// TIA Portal V18 export
// export: Created 2026-06-23T08:49:31.4351033Z, ExportSetting WithDefaults, DisplayName Totally Integrated Automation Portal, DisplayVersion V18, DisplayName TIA Portal Openness, DisplayVersion V18, DisplayName TIA Portal Version Control Interface, DisplayVersion V18, DisplayName STEP 7 Professional, DisplayVersion V18, DisplayName STEP 7 Safety, DisplayVersion V18, DisplayName WinCC Professional, DisplayVersion V18
FUNCTION "FC_HMI_Mirror_PLC2" : Void   // FC41, LAD
{ S7_Optimized_Access := 'TRUE' }
VERSION : 0.1
// stored: AutoNumber true, IsIECCheckEnabled false, SetENOAutomatically false, UDAEnableTagReadback false
BEGIN

REGION Network 1: Mirror V3240_Nuoc_Bon3
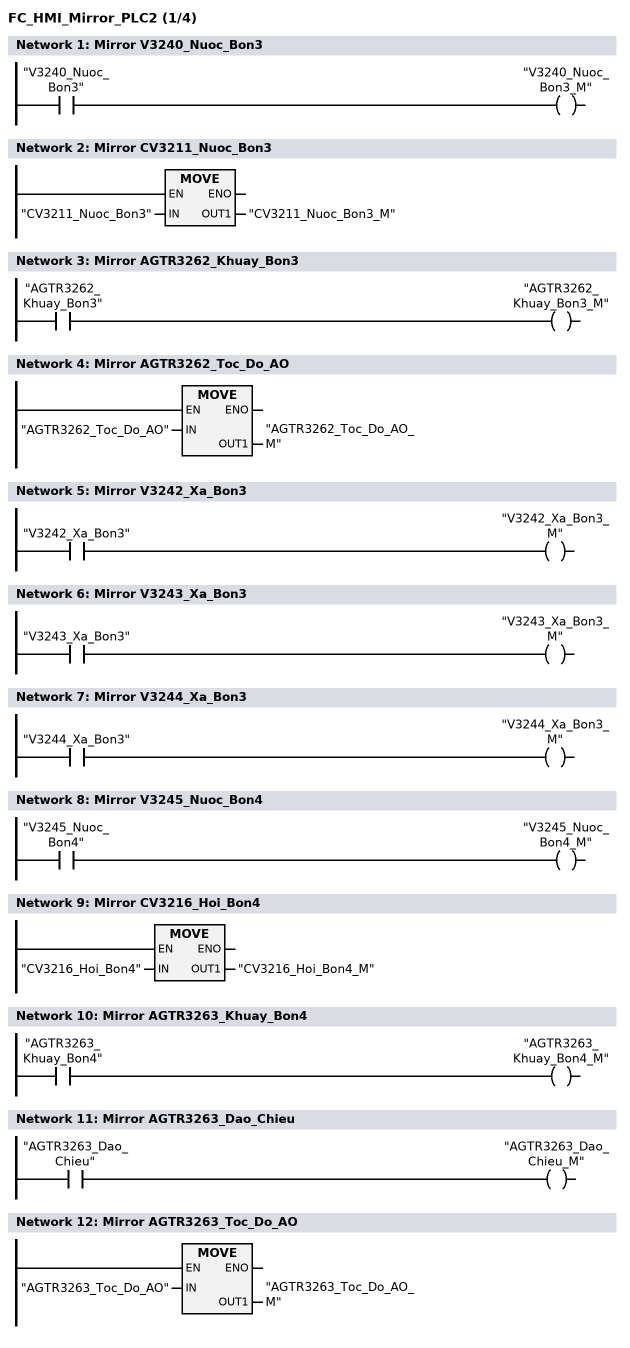
   RUNG wire#powerrail
      Contact( "V3240_Nuoc_Bon3" )
      Coil( "V3240_Nuoc_Bon3_M" )
   END_RUNG
   // the same network as SCL:
   "V3240_Nuoc_Bon3_M" := "V3240_Nuoc_Bon3";
END_REGION

REGION Network 2: Mirror CV3211_Nuoc_Bon3
   RUNG wire#powerrail
      { S7_GenerateENO := "TRUE" } Move(in := "CV3211_Nuoc_Bon3", out1 => "CV3211_Nuoc_Bon3_M")
   END_RUNG
   // the same network as SCL:
   "CV3211_Nuoc_Bon3_M" := "CV3211_Nuoc_Bon3";
END_REGION

REGION Network 3: Mirror AGTR3262_Khuay_Bon3
   RUNG wire#powerrail
      Contact( "AGTR3262_Khuay_Bon3" )
      Coil( "AGTR3262_Khuay_Bon3_M" )
   END_RUNG
   // the same network as SCL:
   "AGTR3262_Khuay_Bon3_M" := "AGTR3262_Khuay_Bon3";
END_REGION

REGION Network 4: Mirror AGTR3262_Toc_Do_AO
   RUNG wire#powerrail
      { S7_GenerateENO := "TRUE" } Move(in := "AGTR3262_Toc_Do_AO", out1 => "AGTR3262_Toc_Do_AO_M")
   END_RUNG
   // the same network as SCL:
   "AGTR3262_Toc_Do_AO_M" := "AGTR3262_Toc_Do_AO";
END_REGION

REGION Network 5: Mirror V3242_Xa_Bon3
   RUNG wire#powerrail
      Contact( "V3242_Xa_Bon3" )
      Coil( "V3242_Xa_Bon3_M" )
   END_RUNG
   // the same network as SCL:
   "V3242_Xa_Bon3_M" := "V3242_Xa_Bon3";
END_REGION

REGION Network 6: Mirror V3243_Xa_Bon3
   RUNG wire#powerrail
      Contact( "V3243_Xa_Bon3" )
      Coil( "V3243_Xa_Bon3_M" )
   END_RUNG
   // the same network as SCL:
   "V3243_Xa_Bon3_M" := "V3243_Xa_Bon3";
END_REGION

REGION Network 7: Mirror V3244_Xa_Bon3
   RUNG wire#powerrail
      Contact( "V3244_Xa_Bon3" )
      Coil( "V3244_Xa_Bon3_M" )
   END_RUNG
   // the same network as SCL:
   "V3244_Xa_Bon3_M" := "V3244_Xa_Bon3";
END_REGION

REGION Network 8: Mirror V3245_Nuoc_Bon4
   RUNG wire#powerrail
      Contact( "V3245_Nuoc_Bon4" )
      Coil( "V3245_Nuoc_Bon4_M" )
   END_RUNG
   // the same network as SCL:
   "V3245_Nuoc_Bon4_M" := "V3245_Nuoc_Bon4";
END_REGION

REGION Network 9: Mirror CV3216_Hoi_Bon4
   RUNG wire#powerrail
      { S7_GenerateENO := "TRUE" } Move(in := "CV3216_Hoi_Bon4", out1 => "CV3216_Hoi_Bon4_M")
   END_RUNG
   // the same network as SCL:
   "CV3216_Hoi_Bon4_M" := "CV3216_Hoi_Bon4";
END_REGION

REGION Network 10: Mirror AGTR3263_Khuay_Bon4
   RUNG wire#powerrail
      Contact( "AGTR3263_Khuay_Bon4" )
      Coil( "AGTR3263_Khuay_Bon4_M" )
   END_RUNG
   // the same network as SCL:
   "AGTR3263_Khuay_Bon4_M" := "AGTR3263_Khuay_Bon4";
END_REGION

REGION Network 11: Mirror AGTR3263_Dao_Chieu
   RUNG wire#powerrail
      Contact( "AGTR3263_Dao_Chieu" )
      Coil( "AGTR3263_Dao_Chieu_M" )
   END_RUNG
   // the same network as SCL:
   "AGTR3263_Dao_Chieu_M" := "AGTR3263_Dao_Chieu";
END_REGION

REGION Network 12: Mirror AGTR3263_Toc_Do_AO
   RUNG wire#powerrail
      { S7_GenerateENO := "TRUE" } Move(in := "AGTR3263_Toc_Do_AO", out1 => "AGTR3263_Toc_Do_AO_M")
   END_RUNG
   // the same network as SCL:
   "AGTR3263_Toc_Do_AO_M" := "AGTR3263_Toc_Do_AO";
END_REGION

REGION Network 13: Mirror V3247_Xa_Bon4
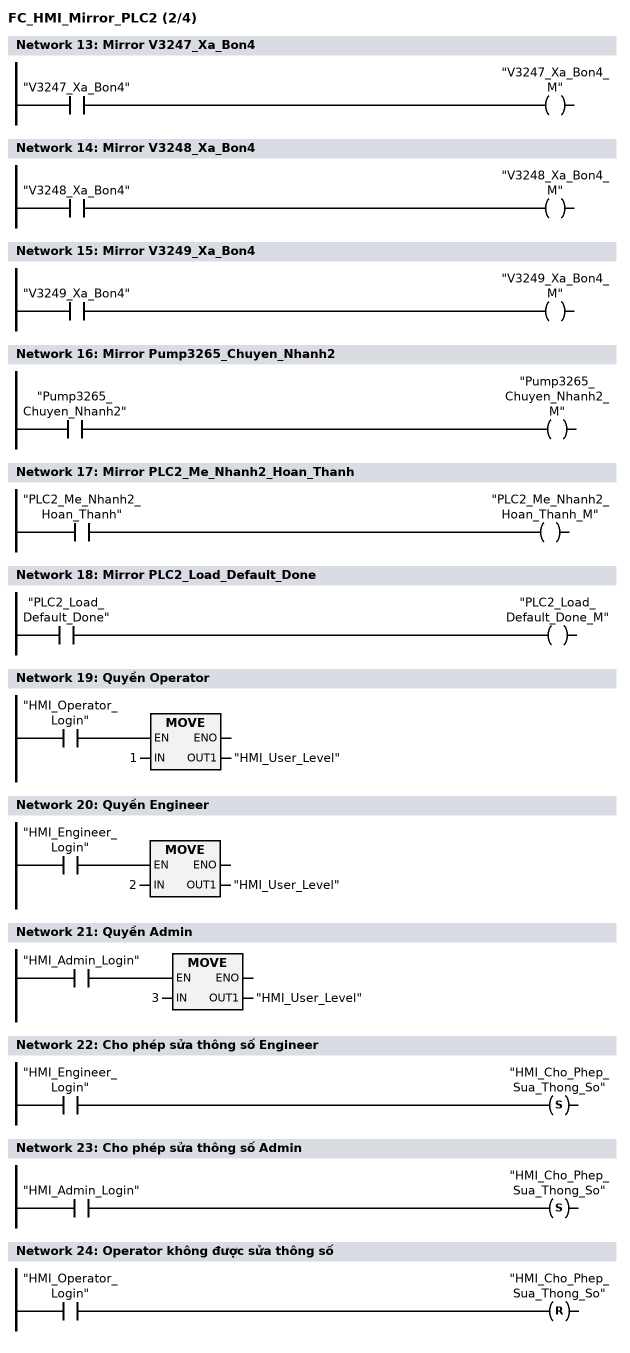
   RUNG wire#powerrail
      Contact( "V3247_Xa_Bon4" )
      Coil( "V3247_Xa_Bon4_M" )
   END_RUNG
   // the same network as SCL:
   "V3247_Xa_Bon4_M" := "V3247_Xa_Bon4";
END_REGION

REGION Network 14: Mirror V3248_Xa_Bon4
   RUNG wire#powerrail
      Contact( "V3248_Xa_Bon4" )
      Coil( "V3248_Xa_Bon4_M" )
   END_RUNG
   // the same network as SCL:
   "V3248_Xa_Bon4_M" := "V3248_Xa_Bon4";
END_REGION

REGION Network 15: Mirror V3249_Xa_Bon4
   RUNG wire#powerrail
      Contact( "V3249_Xa_Bon4" )
      Coil( "V3249_Xa_Bon4_M" )
   END_RUNG
   // the same network as SCL:
   "V3249_Xa_Bon4_M" := "V3249_Xa_Bon4";
END_REGION

REGION Network 16: Mirror Pump3265_Chuyen_Nhanh2
   RUNG wire#powerrail
      Contact( "Pump3265_Chuyen_Nhanh2" )
      Coil( "Pump3265_Chuyen_Nhanh2_M" )
   END_RUNG
   // the same network as SCL:
   "Pump3265_Chuyen_Nhanh2_M" := "Pump3265_Chuyen_Nhanh2";
END_REGION

REGION Network 17: Mirror PLC2_Me_Nhanh2_Hoan_Thanh
   RUNG wire#powerrail
      Contact( "PLC2_Me_Nhanh2_Hoan_Thanh" )
      Coil( "PLC2_Me_Nhanh2_Hoan_Thanh_M" )
   END_RUNG
   // the same network as SCL:
   "PLC2_Me_Nhanh2_Hoan_Thanh_M" := "PLC2_Me_Nhanh2_Hoan_Thanh";
END_REGION

REGION Network 18: Mirror PLC2_Load_Default_Done
   RUNG wire#powerrail
      Contact( "PLC2_Load_Default_Done" )
      Coil( "PLC2_Load_Default_Done_M" )
   END_RUNG
   // the same network as SCL:
   "PLC2_Load_Default_Done_M" := "PLC2_Load_Default_Done";
END_REGION

REGION Network 19: Quyền Operator
   RUNG wire#powerrail
      Contact( "HMI_Operator_Login" )
      { S7_GenerateENO := "TRUE" } Move(in := 1, out1 => "HMI_User_Level")
   END_RUNG
   // the same network as SCL:
   IF "HMI_Operator_Login" THEN "HMI_User_Level" := 1; END_IF;
END_REGION

REGION Network 20: Quyền Engineer
   RUNG wire#powerrail
      Contact( "HMI_Engineer_Login" )
      { S7_GenerateENO := "TRUE" } Move(in := 2, out1 => "HMI_User_Level")
   END_RUNG
   // the same network as SCL:
   IF "HMI_Engineer_Login" THEN "HMI_User_Level" := 2; END_IF;
END_REGION

REGION Network 21: Quyền Admin
   RUNG wire#powerrail
      Contact( "HMI_Admin_Login" )
      { S7_GenerateENO := "TRUE" } Move(in := 3, out1 => "HMI_User_Level")
   END_RUNG
   // the same network as SCL:
   IF "HMI_Admin_Login" THEN "HMI_User_Level" := 3; END_IF;
END_REGION

REGION Network 22: Cho phép sửa thông số Engineer
   RUNG wire#powerrail
      Contact( "HMI_Engineer_Login" )
      S_Coil( "HMI_Cho_Phep_Sua_Thong_So" )
   END_RUNG
   // the same network as SCL:
   IF "HMI_Engineer_Login" THEN "HMI_Cho_Phep_Sua_Thong_So" := TRUE; END_IF;
END_REGION

REGION Network 23: Cho phép sửa thông số Admin
   RUNG wire#powerrail
      Contact( "HMI_Admin_Login" )
      S_Coil( "HMI_Cho_Phep_Sua_Thong_So" )
   END_RUNG
   // the same network as SCL:
   IF "HMI_Admin_Login" THEN "HMI_Cho_Phep_Sua_Thong_So" := TRUE; END_IF;
END_REGION

REGION Network 24: Operator không được sửa thông số
   RUNG wire#powerrail
      Contact( "HMI_Operator_Login" )
      R_Coil( "HMI_Cho_Phep_Sua_Thong_So" )
   END_RUNG
   // the same network as SCL:
   IF "HMI_Operator_Login" THEN "HMI_Cho_Phep_Sua_Thong_So" := FALSE; END_IF;
END_REGION

REGION Network 25: Mã an toàn mặc định
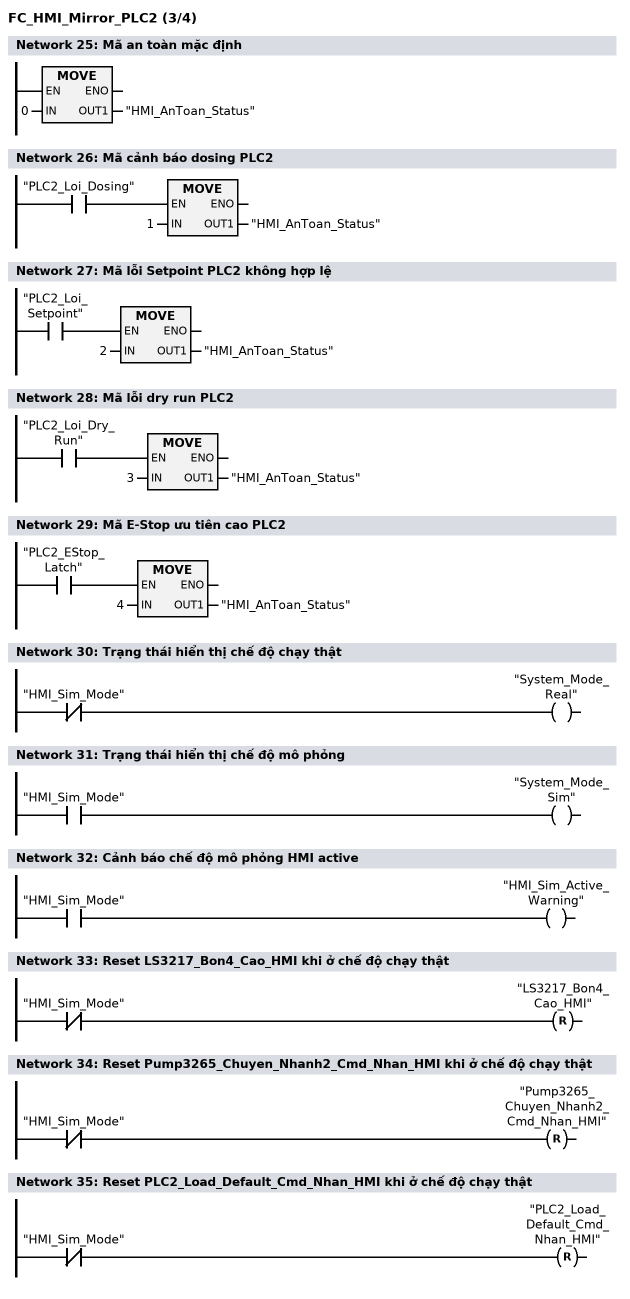
   RUNG wire#powerrail
      { S7_GenerateENO := "TRUE" } Move(in := 0, out1 => "HMI_AnToan_Status")
   END_RUNG
   // the same network as SCL:
   "HMI_AnToan_Status" := 0;
END_REGION

REGION Network 26: Mã cảnh báo dosing PLC2
   RUNG wire#powerrail
      Contact( "PLC2_Loi_Dosing" )
      { S7_GenerateENO := "TRUE" } Move(in := 1, out1 => "HMI_AnToan_Status")
   END_RUNG
   // the same network as SCL:
   IF "PLC2_Loi_Dosing" THEN "HMI_AnToan_Status" := 1; END_IF;
END_REGION

REGION Network 27: Mã lỗi Setpoint PLC2 không hợp lệ
   RUNG wire#powerrail
      Contact( "PLC2_Loi_Setpoint" )
      { S7_GenerateENO := "TRUE" } Move(in := 2, out1 => "HMI_AnToan_Status")
   END_RUNG
   // the same network as SCL:
   IF "PLC2_Loi_Setpoint" THEN "HMI_AnToan_Status" := 2; END_IF;
END_REGION

REGION Network 28: Mã lỗi dry run PLC2
   RUNG wire#powerrail
      Contact( "PLC2_Loi_Dry_Run" )
      { S7_GenerateENO := "TRUE" } Move(in := 3, out1 => "HMI_AnToan_Status")
   END_RUNG
   // the same network as SCL:
   IF "PLC2_Loi_Dry_Run" THEN "HMI_AnToan_Status" := 3; END_IF;
END_REGION

REGION Network 29: Mã E-Stop ưu tiên cao PLC2
   RUNG wire#powerrail
      Contact( "PLC2_EStop_Latch" )
      { S7_GenerateENO := "TRUE" } Move(in := 4, out1 => "HMI_AnToan_Status")
   END_RUNG
   // the same network as SCL:
   IF "PLC2_EStop_Latch" THEN "HMI_AnToan_Status" := 4; END_IF;
END_REGION

REGION Network 30: Trạng thái hiển thị chế độ chạy thật
   RUNG wire#powerrail
      I_Contact( "HMI_Sim_Mode" )
      Coil( "System_Mode_Real" )
   END_RUNG
   // the same network as SCL:
   "System_Mode_Real" := NOT "HMI_Sim_Mode";
END_REGION

REGION Network 31: Trạng thái hiển thị chế độ mô phỏng
   RUNG wire#powerrail
      Contact( "HMI_Sim_Mode" )
      Coil( "System_Mode_Sim" )
   END_RUNG
   // the same network as SCL:
   "System_Mode_Sim" := "HMI_Sim_Mode";
END_REGION

REGION Network 32: Cảnh báo chế độ mô phỏng HMI active
   RUNG wire#powerrail
      Contact( "HMI_Sim_Mode" )
      Coil( "HMI_Sim_Active_Warning" )
   END_RUNG
   // the same network as SCL:
   "HMI_Sim_Active_Warning" := "HMI_Sim_Mode";
END_REGION

REGION Network 33: Reset LS3217_Bon4_Cao_HMI khi ở chế độ chạy thật
   RUNG wire#powerrail
      I_Contact( "HMI_Sim_Mode" )
      R_Coil( "LS3217_Bon4_Cao_HMI" )
   END_RUNG
   // the same network as SCL:
   IF NOT "HMI_Sim_Mode" THEN "LS3217_Bon4_Cao_HMI" := FALSE; END_IF;
END_REGION

REGION Network 34: Reset Pump3265_Chuyen_Nhanh2_Cmd_Nhan_HMI khi ở chế độ chạy thật
   RUNG wire#powerrail
      I_Contact( "HMI_Sim_Mode" )
      R_Coil( "Pump3265_Chuyen_Nhanh2_Cmd_Nhan_HMI" )
   END_RUNG
   // the same network as SCL:
   IF NOT "HMI_Sim_Mode" THEN "Pump3265_Chuyen_Nhanh2_Cmd_Nhan_HMI" := FALSE; END_IF;
END_REGION

REGION Network 35: Reset PLC2_Load_Default_Cmd_Nhan_HMI khi ở chế độ chạy thật
   RUNG wire#powerrail
      I_Contact( "HMI_Sim_Mode" )
      R_Coil( "PLC2_Load_Default_Cmd_Nhan_HMI" )
   END_RUNG
   // the same network as SCL:
   IF NOT "HMI_Sim_Mode" THEN "PLC2_Load_Default_Cmd_Nhan_HMI" := FALSE; END_IF;
END_REGION

REGION Network 36: Reset FT3210_Bon3_HMI về 0.0 khi ở chế độ chạy thật
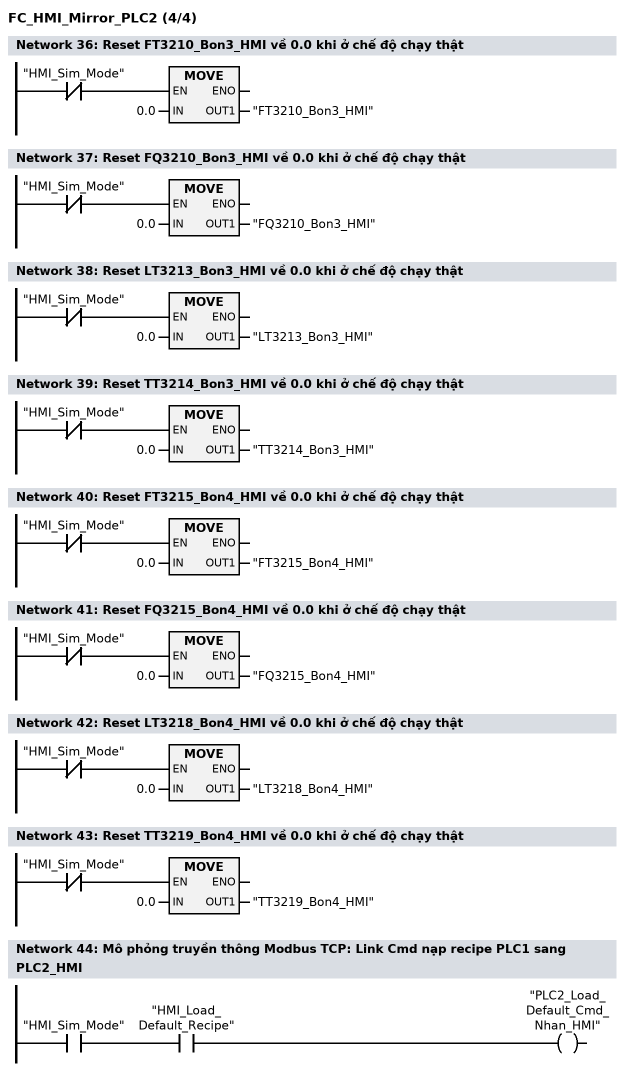
   RUNG wire#powerrail
      I_Contact( "HMI_Sim_Mode" )
      { S7_GenerateENO := "TRUE" } Move(in := 0.0, out1 => "FT3210_Bon3_HMI")
   END_RUNG
   // the same network as SCL:
   IF NOT "HMI_Sim_Mode" THEN "FT3210_Bon3_HMI" := 0.0; END_IF;
END_REGION

REGION Network 37: Reset FQ3210_Bon3_HMI về 0.0 khi ở chế độ chạy thật
   RUNG wire#powerrail
      I_Contact( "HMI_Sim_Mode" )
      { S7_GenerateENO := "TRUE" } Move(in := 0.0, out1 => "FQ3210_Bon3_HMI")
   END_RUNG
   // the same network as SCL:
   IF NOT "HMI_Sim_Mode" THEN "FQ3210_Bon3_HMI" := 0.0; END_IF;
END_REGION

REGION Network 38: Reset LT3213_Bon3_HMI về 0.0 khi ở chế độ chạy thật
   RUNG wire#powerrail
      I_Contact( "HMI_Sim_Mode" )
      { S7_GenerateENO := "TRUE" } Move(in := 0.0, out1 => "LT3213_Bon3_HMI")
   END_RUNG
   // the same network as SCL:
   IF NOT "HMI_Sim_Mode" THEN "LT3213_Bon3_HMI" := 0.0; END_IF;
END_REGION

REGION Network 39: Reset TT3214_Bon3_HMI về 0.0 khi ở chế độ chạy thật
   RUNG wire#powerrail
      I_Contact( "HMI_Sim_Mode" )
      { S7_GenerateENO := "TRUE" } Move(in := 0.0, out1 => "TT3214_Bon3_HMI")
   END_RUNG
   // the same network as SCL:
   IF NOT "HMI_Sim_Mode" THEN "TT3214_Bon3_HMI" := 0.0; END_IF;
END_REGION

REGION Network 40: Reset FT3215_Bon4_HMI về 0.0 khi ở chế độ chạy thật
   RUNG wire#powerrail
      I_Contact( "HMI_Sim_Mode" )
      { S7_GenerateENO := "TRUE" } Move(in := 0.0, out1 => "FT3215_Bon4_HMI")
   END_RUNG
   // the same network as SCL:
   IF NOT "HMI_Sim_Mode" THEN "FT3215_Bon4_HMI" := 0.0; END_IF;
END_REGION

REGION Network 41: Reset FQ3215_Bon4_HMI về 0.0 khi ở chế độ chạy thật
   RUNG wire#powerrail
      I_Contact( "HMI_Sim_Mode" )
      { S7_GenerateENO := "TRUE" } Move(in := 0.0, out1 => "FQ3215_Bon4_HMI")
   END_RUNG
   // the same network as SCL:
   IF NOT "HMI_Sim_Mode" THEN "FQ3215_Bon4_HMI" := 0.0; END_IF;
END_REGION

REGION Network 42: Reset LT3218_Bon4_HMI về 0.0 khi ở chế độ chạy thật
   RUNG wire#powerrail
      I_Contact( "HMI_Sim_Mode" )
      { S7_GenerateENO := "TRUE" } Move(in := 0.0, out1 => "LT3218_Bon4_HMI")
   END_RUNG
   // the same network as SCL:
   IF NOT "HMI_Sim_Mode" THEN "LT3218_Bon4_HMI" := 0.0; END_IF;
END_REGION

REGION Network 43: Reset TT3219_Bon4_HMI về 0.0 khi ở chế độ chạy thật
   RUNG wire#powerrail
      I_Contact( "HMI_Sim_Mode" )
      { S7_GenerateENO := "TRUE" } Move(in := 0.0, out1 => "TT3219_Bon4_HMI")
   END_RUNG
   // the same network as SCL:
   IF NOT "HMI_Sim_Mode" THEN "TT3219_Bon4_HMI" := 0.0; END_IF;
END_REGION

REGION Network 44: Mô phỏng truyền thông Modbus TCP: Link Cmd nạp recipe PLC1 sang PLC2_HMI
   RUNG wire#powerrail
      Contact( "HMI_Sim_Mode" )
      Contact( "HMI_Load_Default_Recipe" )
      Coil( "PLC2_Load_Default_Cmd_Nhan_HMI" )
   END_RUNG
   // the same network as SCL:
   "PLC2_Load_Default_Cmd_Nhan_HMI" := "HMI_Sim_Mode" AND "HMI_Load_Default_Recipe";
END_REGION
END_FUNCTION
